TYPE (* DataPanel Modules with medium IO density DO Struct + Source Address *)
  (* Version 1.0, 2026-05-28, franz *)
  PACKAGE DataPanel::io::MI::DQ;
  IMPORT DataPanel::io::MI::const::MI::MI_00;
  IMPORT DataPanel::io::MI::DQ::DataPanel_MI_DO_S;
  IMPORT DataPanel::io::MI::DQ::DataPanel_MI_DO::Invalid;
  DataPanel_MI_DO_S_Octal_SA : STRUCT
    u8SAMember : USINT := MI_00; (* Node SA 224..239 *)
    Port1 : DataPanel::io::MI::DQ::DataPanel_MI_DO_S := Invalid; (* Identify the Port 1A..8B *)
    Port2 : DataPanel::io::MI::DQ::DataPanel_MI_DO_S := Invalid; (* Identify the Port 1A..8B *)
    Port3 : DataPanel::io::MI::DQ::DataPanel_MI_DO_S := Invalid; (* Identify the Port 1A..8B *)
    Port4 : DataPanel::io::MI::DQ::DataPanel_MI_DO_S := Invalid; (* Identify the Port 1A..8B *)
    Port5 : DataPanel::io::MI::DQ::DataPanel_MI_DO_S := Invalid; (* Identify the Port 1A..8B *)
    Port6 : DataPanel::io::MI::DQ::DataPanel_MI_DO_S := Invalid; (* Identify the Port 1A..8B *)
    Port7 : DataPanel::io::MI::DQ::DataPanel_MI_DO_S := Invalid; (* Identify the Port 1A..8B *)
    Port8 : DataPanel::io::MI::DQ::DataPanel_MI_DO_S := Invalid; (* Identify the Port 1A..8B *)
  END_STRUCT;
END_TYPE
